PROGRAM MAIN
VAR
END_VAR

IF TwinCAT_SystemInfoVarList._TaskInfo[GETCURTASKINDEXEX()].FirstCycle THEN
	// For Remote Log4TC Server change the AMS net ID and configure a route
	PRG_TaskLog.Init('127.0.0.1.1.1');
	F_Log(E_LogLevel.eInfo, 'F_Log');
END_IF


PRG_TaskLog.Call();

END_PROGRAM

(* stored: Version 1.1.0.1, ProductVersion 3.1.4024.0
   POU MAIN: Id {8e76aa5e-29ea-465d-a10c-8a373442d35f}, SpecialFunc None *)
